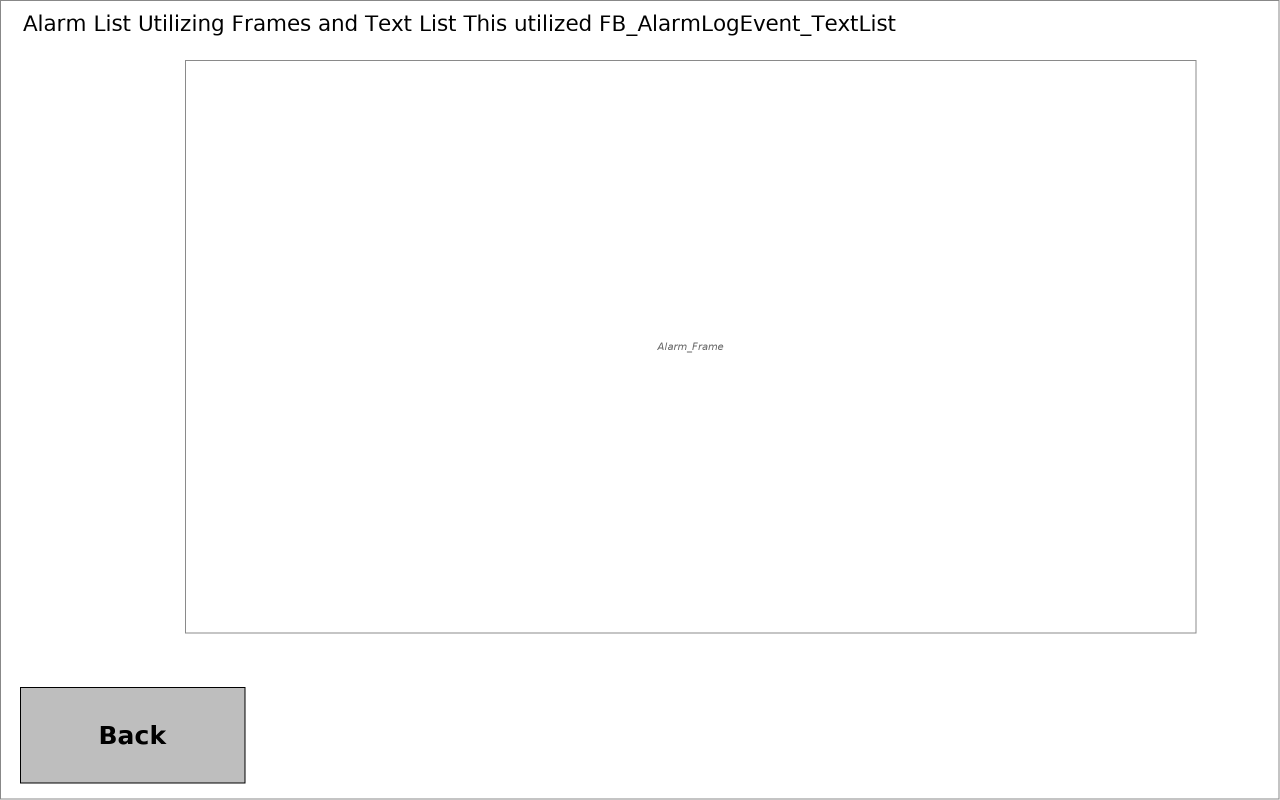
VISUALIZATION Alarms  // 1280x800
    Rectangle (20,9 909x60), "Alarm List Utilizing Frames and Text List This utilized FB_AlarmLogEvent_TextList"
    Frame (185,60 1011x573)
        shows Alarm_Frame(xFaultResetPB := HMI.xFaultResetPB, sAlarmTextList := 'Alarm_TextList', sEventDataTextList := 'stAlarmEventData_TextList', astActiveAlarmsList_1 := HMI.astActiveAlarmsList[1], astActiveAlarmsList_2 := HMI.astActiveAlarmsList[2], astActiveAlarmsList_3 := HMI.astActiveAlarmsList[3], astActiveAlarmsList_4 := HMI.astActiveAlarmsList[4], astActiveAlarmsList_5 := HMI.astActiveAlarmsList[5], astActiveAlarmsList_6 := HMI.astActiveAlarmsList[6], astActiveAlarmsList_7 := HMI.astActiveAlarmsList[7], astActiveAlarmsList_8 := HMI.astActiveAlarmsList[8])
    Rectangle (20,687 225x96), "Back"
        OnMouseClick: change screen: Previous Alarm_Table
END_VISUALIZATION

(* stored: Version 1.1.0.1
   Visu Alarms: Id {4af80912-0288-4990-887a-58ee8c532c07} *)
